FUNCTION_BLOCK CallbackFB (* Composite FB wrapping other FBs *)
  (* Standard: 61499-2 *)
  (* Version 1.0, 2025-09-06, franz *)
  PACKAGE isobus::tx;
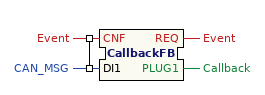
  EVENT_INPUT
    CNF WITH DI1; (* Confirmation from Plug *)
  END_EVENT
  EVENT_OUTPUT
    REQ; (* Request from Socket *)
  END_EVENT
  VAR_INPUT
    DI1 : isobus::CAN_MSG;
  END_VAR
  PLUGS
    PLUG1 : isobus::tx::Callback;
  END_PLUGS
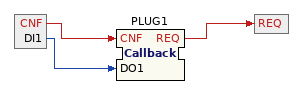
  EVENT_CONNECTIONS
    CNF TO PLUG1.CNF;
    PLUG1.REQ TO REQ;
  END_CONNECTIONS
  DATA_CONNECTIONS
    DI1 TO PLUG1.DO1;
  END_CONNECTIONS
END_FUNCTION_BLOCK
